RoboDK station: 圆形D400mm_v50.rdk

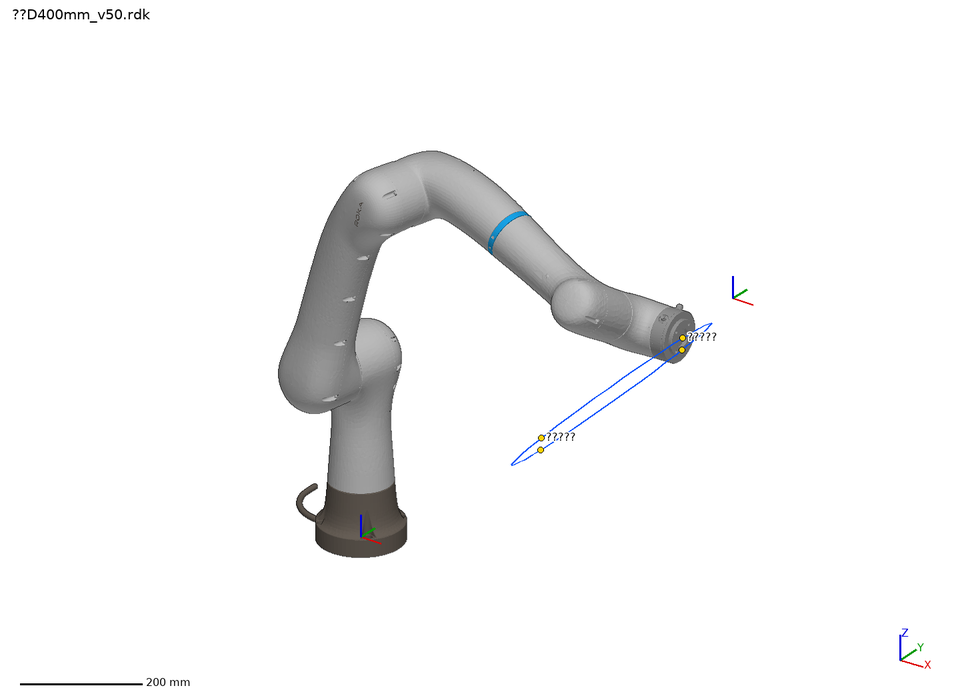
[picture v0: the station drawn from its stored meshes, robots at their saved joint values, targets as dots, program paths as lines]
Station 圆形D400mm_v50 (saved by RoboDK 5.9.0). Poses are relative to the parent item; angles as X-Y-Z fixed-axis rotations.
  - frame Rokae SR4-C Base at (0, 0, 0) mm
    - robot Rokae SR4-C: 6 axes
        modified DH rows (alpha deg, a mm, theta deg, d mm): 0, 0, 0, 328; -90, 0, -82.875, 0; 0, 400, -97.125, 0; -90, 50, 0, 400; 90, 0, 0, 136; -90, 0, 180, 103.5
        joint limits [-360, -160, -170, -200, -360, -360] to [360, 150, 140, 360, 360, 360]; home [0, 0, -90, 0, 0, 0]; saved at [-12.195, 15.853, -93.337, -33.325, 22.613, 31.256]
      - tool Tool 1, TCP at (0, 0, 0) mm
    - frame 大圆运动坐标系 at (741.44, 0, 641.44) mm
      - target 大圆上顶点 (Cartesian target) at (-100, 0, -100) mm, rotated rx 0 ry 90 rz 0 deg; joints [-12.195, 15.853, -93.337, -33.325, 22.613, 31.256] of Rokae SR4-C
      - target 大圆左顶点 (Cartesian target) at (-241.44, -200, -241.44) mm, rotated rx 0 ry 90 rz 0 deg; joints [-37.866, 16.402, -112.53, -51.054, 52.113, 37.228] of Rokae SR4-C
      - target 大圆下顶点 (Cartesian target) at (-382.88, 0, -382.88) mm, rotated rx 0 ry 90 rz 0 deg; joints [-28.064, 27.082, -150.883, -28.079, 88.205, 0.958] of Rokae SR4-C
      - target 大圆右顶点 (Cartesian target) at (-241.44, 200, -241.44) mm, rotated rx 0 ry 90 rz 0 deg; joints [9.265, 14.582, -133.523, 10.876, 58.57, -5.721] of Rokae SR4-C
  - program 程序1 (6 instructions, listed below)

--- program 程序1 (robot Rokae SR4-C) ---
  设置参考: 大圆运动坐标系
  设置工具: Tool 1
  MoveJ (大圆上顶点)
  设置速度（50.0 mm/s)
  MoveC (大圆右顶点, 大圆下顶点)
  MoveC (大圆左顶点, 大圆上顶点)
